# EPICS substitutions: icpdasApp/Db/icp7026.substitutions
file "icpai.template"
{
    pattern {P,     R,   REGOFFSET, PORT,   }
            {$(P),  $(R),     0,         $(AIPORT)}
            {$(P),  $(R),     1,         $(AIPORT)}
            {$(P),  $(R),     2,         $(AIPORT)}
            {$(P),  $(R),     3,         $(AIPORT)}
            {$(P),  $(R),     4,         $(AIPORT)}
            {$(P),  $(R),     5,         $(AIPORT)}

}

file "icpao.template"
{
    pattern {P,     R,   REGOFFSET, PORT,   PORTRB}
            {$(P),  $(R),     0,         $(AOPORT), $(AOPORTRB)  }
            {$(P),  $(R),     1,         $(AOPORT), $(AOPORTRB)  }
}

file "icpdi.template"
{
    pattern {P,     R,   REGOFFSET, PORT,   }
            {$(P),  $(R),     0,         $(AIPORT)}
            {$(P),  $(R),     1,         $(AIPORT)}
}

file "icpdo.template"
{
    pattern {P,     R,   REGOFFSET, PORT,   PORTRB}
            {$(P),  $(R),     0,         $(AOPORT), $(AOPORTRB)  }
            {$(P),  $(R),     1,         $(AOPORT), $(AOPORTRB)  }
}
